Staubli VAL3: Main.pgx

public program Main()
  local num l_nKey
begin
  //
  bUserRefresh=bListRefresh=true
  bExit=false
  //
  do
    call Refresh()
    call RefreshList()
    call user:setList("",sList,bUserRefresh,bListRefresh,nSelected,sItem,l_nKey)
    bUserRefresh=false
    bListRefresh=false
    call MainKey(l_nKey)
    delay(0)
  until bExit

end
